FUNCTION_BLOCK ABSTRACT FB_AirConditionerBase EXTENDS FB_Device
VAR_INPUT
END_VAR
VAR_OUTPUT
END_VAR
VAR
END_VAR

METHOD TurnOff : BOOL
VAR_INPUT
END_VAR
END_METHOD

METHOD TurnOn : BOOL
VAR_INPUT
END_VAR
END_METHOD

END_FUNCTION_BLOCK

(* stored: Version 1.1.0.1, ProductVersion 3.1.4024.9
   POU FB_AirConditionerBase: Id {8a14cb96-ec1e-44a6-964e-020b0d9869d0}, SpecialFunc None
   Method TurnOff: Id {63713da6-a9b0-4c78-8811-764f20c72265}
   Method TurnOn: Id {19db32a1-132c-4ed7-96f3-ecd21742b63a} *)
